(*
SPDX-FileCopyrightText: © 2026 Oleksandr Tiutyk <trofimich@gmail.com>
SPDX-License-Identifier: MIT
License: https://opensource.org/license/mit
*)

TYPE ERROR_MESSAGE : WSTRING(2000); END_TYPE

(* stored: Version 1.1.0.1
   DUT ERROR_MESSAGE: Id {72b9ae2b-081e-4ecb-b762-9c7dd5d48450} *)
